TYPE TYP_HW_L4000_OUT :
STRUCT
	AcqCtrl : TYP_HW_L4000_ACQ_CTRL;
	InspCtrl : TYP_HW_L4000_INSP_CTRL;
	CommandID AT %Q* : UINT;
	ExternalEvent : TYP_HW_L4000_EXT_CTRL;
	UserData AT %Q* : ARRAY[0..63] OF BYTE;
END_STRUCT
END_TYPE

(* stored: Version 1.1.0.1, ProductVersion 3.1.4024.12
   DUT TYP_HW_L4000_OUT: Id {4a95c398-d2a7-4901-86a3-21d25f28994b} *)
